// TIA Portal project "Erronka3 Igogailua" (V15.1)

(* hardware
DEVICE "S7-1200 station_1"  S7-1200 Station
   slot 0: "Rack_0"  S7-1200 Rack  Rack  V1.0
   slot 1: "PLC_1"  CPU 1214C AC/DC/Rly  6ES7 214-1BG40-0XB0  V4.2
*)

// ===== PLC "PLC_1"  CPU 1214C AC/DC/Rly =====

VAR_GLOBAL   // PLC tag table "Etapak"
   "Etapa0" AT %M16.0 : Bool;
   "Etapa1" AT %M16.1 : Bool;
   "Etapa2" AT %M16.2 : Bool;
   "Etapa3" AT %M16.3 : Bool;
   "Etapa4" AT %M16.4 : Bool;
   "Etapa5" AT %M16.5 : Bool;
   "Etapa6" AT %M16.6 : Bool;
   "Etapa3.1" AT %M17.0 : Bool;
   "Etapa10" AT %M17.1 : Bool;
   "Etapa11" AT %M17.2 : Bool;
   "Etapa12" AT %M17.3 : Bool;
   "Etapa13" AT %M17.4 : Bool;
   "Etapa14" AT %M17.5 : Bool;
   "Etapa11.1" AT %M17.6 : Bool;
   "Etapa40" AT %M17.7 : Bool;
   "Etapa41" AT %M18.0 : Bool;
   "Etapa42" AT %M18.1 : Bool;
   "Etapa43" AT %M18.2 : Bool;
   "Etapa44" AT %M18.3 : Bool;
   "Etapa50" AT %M18.4 : Bool;
   "Etapa51" AT %M18.5 : Bool;
   "Etapa52" AT %M18.6 : Bool;
   "Etapa53" AT %M18.7 : Bool;
   "Etapa54" AT %M19.0 : Bool;
   "Etapa60" AT %M19.1 : Bool;
   "Etapa61" AT %M19.2 : Bool;
END_VAR

VAR_GLOBAL   // PLC tag table "Irterak"
   "M1Subir" AT %Q0.0 : Bool;
   "M2Abrir" AT %Q0.1 : Bool;
   "M1Bajar" AT %Q0.2 : Bool;
   "M2Cerrar" AT %Q0.3 : Bool;
   "0Sube" AT %Q0.4 : Bool;
   "0Baja" AT %Q0.5 : Bool;
   "1Sube" AT %Q0.6 : Bool;
   "1Baja" AT %Q0.7 : Bool;
   "ASube" AT %Q1.0 : Bool;
   "ABaja" AT %Q1.1 : Bool;
   "M1Subir_10" AT %Q1.2 : Bool;
END_VAR

VAR_GLOBAL   // PLC tag table "Sarrerak"
   "FC0" AT %I0.0 : Bool;
   "FC1" AT %I0.1 : Bool;
   "PF0" AT %I0.2 : Bool;
   "PF1" AT %I0.3 : Bool;
   "PD1" AT %I0.4 : Bool;
   "PD0" AT %I0.5 : Bool;
   "PA" AT %I0.6 : Bool;
   "F" AT %I0.7 : Bool;
   "M" AT %I1.0 : Bool;
   "SCP" AT %I1.1 : Bool;
   "SAP" AT %I1.2 : Bool;
   "PE" AT %I1.3 : Bool;
END_VAR

// folder: System blocks/Program resources

DATA_BLOCK "Temporizador1"   // DB1
{ S7_Optimized_Access := 'TRUE' }
AUTHOR : Simatic
FAMILY : IEC
NAME : IEC_TMR
VERSION : 1.0
// stored: InstanceOfName IEC_TIMER
"IEC_TIMER"
BEGIN
END_DATA_BLOCK

// folder: (top level)

FUNCTION "Grafcet" : Void   // FC1, LAD
{ S7_Optimized_Access := 'TRUE' }
VERSION : 0.1
BEGIN

REGION Network 1: Activar etapa 1
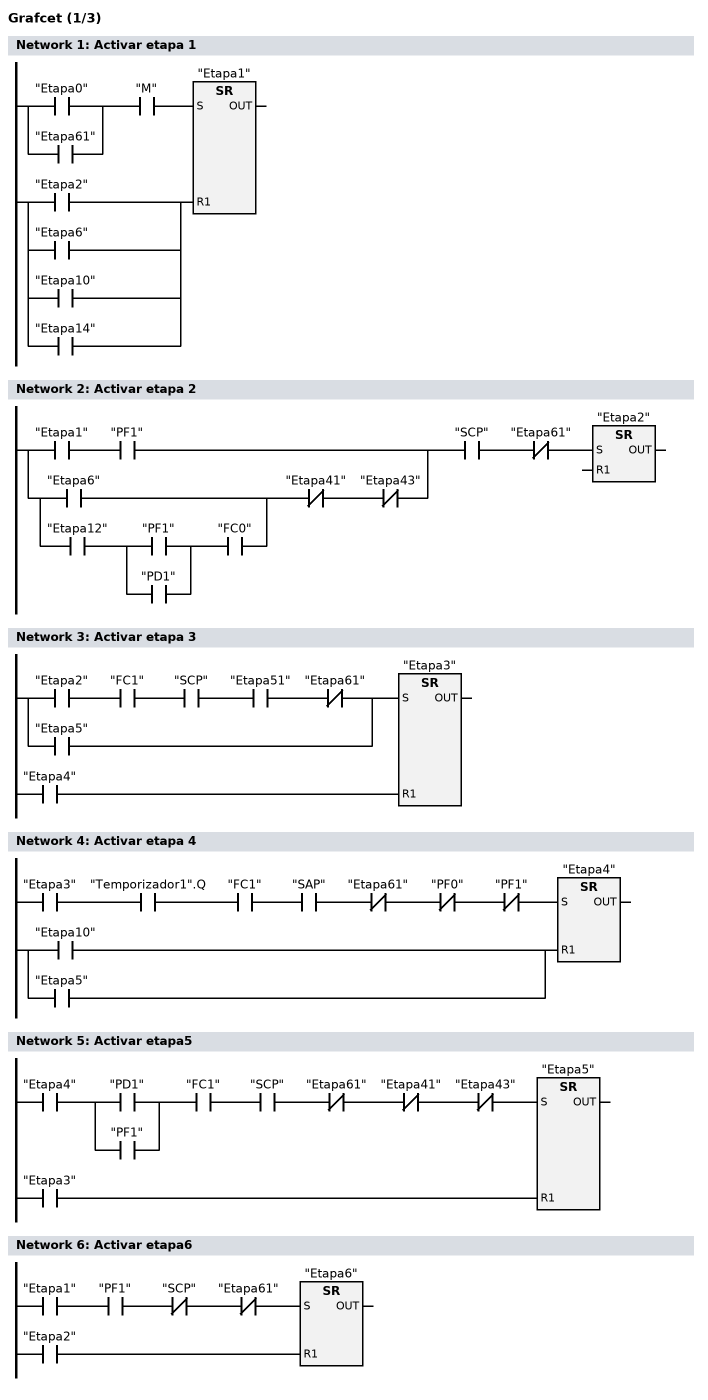
   RUNG wire#powerrail
      Contact( "Etapa0" )
      wire#w1
      Contact( "M" )
      S_SR(operand := "Etapa1", r1 := wire#w2)
   END_RUNG
   RUNG wire#powerrail
      Contact( "Etapa61" )
   END_RUNG wire#w1
   RUNG wire#powerrail
      Contact( "Etapa2" )
   END_RUNG wire#w2
   RUNG wire#powerrail
      Contact( "Etapa6" )
   END_RUNG wire#w2
   RUNG wire#powerrail
      Contact( "Etapa10" )
   END_RUNG wire#w2
   RUNG wire#powerrail
      Contact( "Etapa14" )
   END_RUNG wire#w2
   // the same network as SCL:
   IF ("Etapa0" OR "Etapa61") AND "M" THEN
       "Etapa1" := TRUE;   // SR flip-flop
   END_IF;
   IF "Etapa2" OR "Etapa6" OR "Etapa10" OR "Etapa14" THEN "Etapa1" := FALSE; END_IF;
END_REGION

REGION Network 2: Activar etapa 2
   RUNG wire#powerrail
      Contact( "Etapa1" )
      Contact( "PF1" )
      wire#w1
      Contact( "SCP" )
      I_Contact( "Etapa61" )
      S_SR(operand := "Etapa2", r1 :=)
   END_RUNG
   RUNG wire#powerrail
      Contact( "Etapa6" )
      wire#w2
      I_Contact( "Etapa41" )
      I_Contact( "Etapa43" )
   END_RUNG wire#w1
   RUNG wire#powerrail
      Contact( "Etapa12" )
      wire#w3
      Contact( "PF1" )
      wire#w4
      Contact( "FC0" )
   END_RUNG wire#w2
   RUNG wire#w3
      Contact( "PD1" )
   END_RUNG wire#w4
   // the same network as SCL:
   IF (("Etapa1" AND "PF1") OR (("Etapa6" OR ("Etapa12" AND ("PF1" OR "PD1") AND "FC0")) AND NOT "Etapa41" AND NOT "Etapa43")) AND "SCP" AND NOT "Etapa61" THEN
       "Etapa2" := TRUE;   // SR flip-flop
   END_IF;
END_REGION

REGION Network 3: Activar etapa 3
   RUNG wire#powerrail
      Contact( "Etapa2" )
      Contact( "FC1" )
      Contact( "SCP" )
      Contact( "Etapa51" )
      I_Contact( "Etapa61" )
      wire#w1
      S_SR(operand := "Etapa3", r1 := wire#w2)
   END_RUNG
   RUNG wire#powerrail
      Contact( "Etapa5" )
   END_RUNG wire#w1
   RUNG wire#powerrail
      Contact( "Etapa4" )
   END_RUNG wire#w2
   // the same network as SCL:
   IF ("Etapa2" AND "FC1" AND "SCP" AND "Etapa51" AND NOT "Etapa61") OR "Etapa5" THEN
       "Etapa3" := TRUE;   // SR flip-flop
   END_IF;
   IF "Etapa4" THEN "Etapa3" := FALSE; END_IF;
END_REGION

REGION Network 4: Activar etapa 4
   RUNG wire#powerrail
      Contact( "Etapa3" )
      Contact( "Temporizador1".Q )
      Contact( "FC1" )
      Contact( "SAP" )
      I_Contact( "Etapa61" )
      I_Contact( "PF0" )
      I_Contact( "PF1" )
      S_SR(operand := "Etapa4", r1 := wire#w1)
   END_RUNG
   RUNG wire#powerrail
      Contact( "Etapa10" )
   END_RUNG wire#w1
   RUNG wire#powerrail
      Contact( "Etapa5" )
   END_RUNG wire#w1
   // the same network as SCL:
   IF "Etapa3" AND "Temporizador1".Q AND "FC1" AND "SAP" AND NOT "Etapa61" AND NOT "PF0" AND NOT "PF1" THEN
       "Etapa4" := TRUE;   // SR flip-flop
   END_IF;
   IF "Etapa10" OR "Etapa5" THEN "Etapa4" := FALSE; END_IF;
END_REGION

REGION Network 5: Activar etapa5
   RUNG wire#powerrail
      Contact( "Etapa4" )
      wire#w1
      Contact( "PD1" )
      wire#w2
      Contact( "FC1" )
      Contact( "SCP" )
      I_Contact( "Etapa61" )
      I_Contact( "Etapa41" )
      I_Contact( "Etapa43" )
      S_SR(operand := "Etapa5", r1 := wire#w3)
   END_RUNG
   RUNG wire#w1
      Contact( "PF1" )
   END_RUNG wire#w2
   RUNG wire#powerrail
      Contact( "Etapa3" )
   END_RUNG wire#w3
   // the same network as SCL:
   IF "Etapa4" AND ("PD1" OR "PF1") AND "FC1" AND "SCP" AND NOT "Etapa61" AND NOT "Etapa41" AND NOT "Etapa43" THEN
       "Etapa5" := TRUE;   // SR flip-flop
   END_IF;
   IF "Etapa3" THEN "Etapa5" := FALSE; END_IF;
END_REGION

REGION Network 6: Activar etapa6
   RUNG wire#powerrail
      Contact( "Etapa1" )
      Contact( "PF1" )
      I_Contact( "SCP" )
      I_Contact( "Etapa61" )
      S_SR(operand := "Etapa6", r1 := wire#w1)
   END_RUNG
   RUNG wire#powerrail
      Contact( "Etapa2" )
   END_RUNG wire#w1
   // the same network as SCL:
   IF "Etapa1" AND "PF1" AND NOT "SCP" AND NOT "Etapa61" THEN
       "Etapa6" := TRUE;   // SR flip-flop
   END_IF;
   IF "Etapa2" THEN "Etapa6" := FALSE; END_IF;
END_REGION

REGION Network 7: Activar etapa3.1
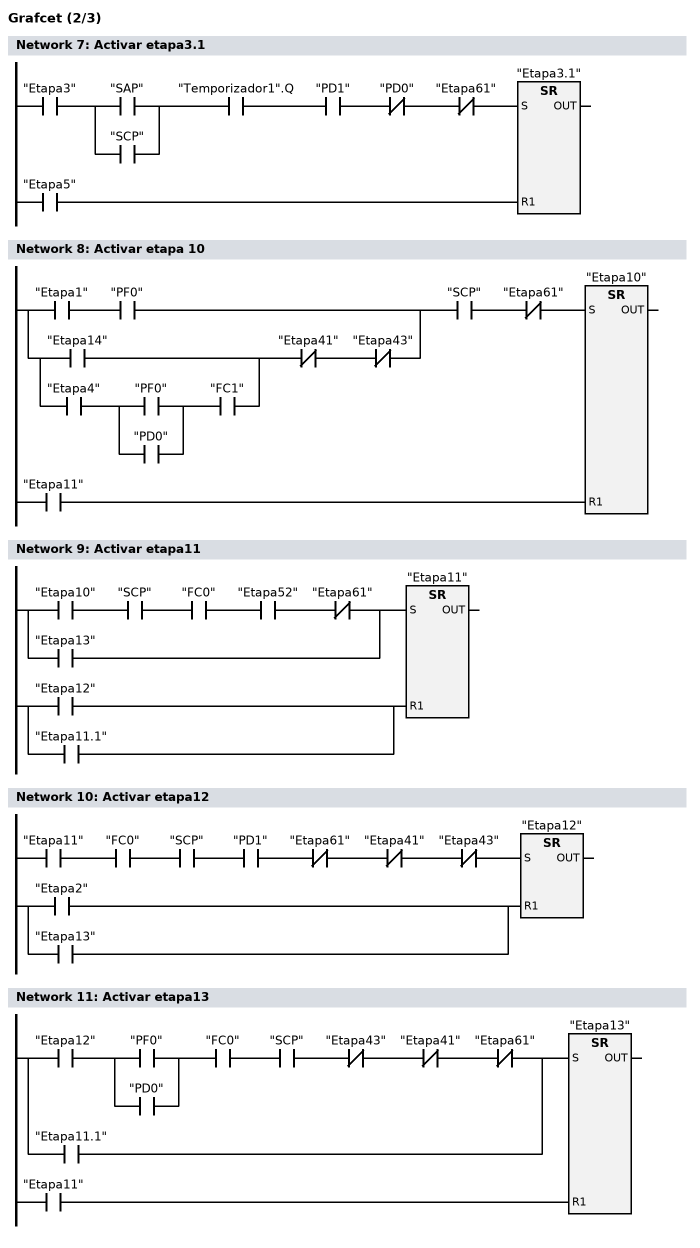
   RUNG wire#powerrail
      Contact( "Etapa3" )
      wire#w1
      Contact( "SAP" )
      wire#w2
      Contact( "Temporizador1".Q )
      Contact( "PD1" )
      I_Contact( "PD0" )
      I_Contact( "Etapa61" )
      S_SR(operand := "Etapa3.1", r1 := wire#w3)
   END_RUNG
   RUNG wire#w1
      Contact( "SCP" )
   END_RUNG wire#w2
   RUNG wire#powerrail
      Contact( "Etapa5" )
   END_RUNG wire#w3
   // the same network as SCL:
   IF "Etapa3" AND ("SAP" OR "SCP") AND "Temporizador1".Q AND "PD1" AND NOT "PD0" AND NOT "Etapa61" THEN
       "Etapa3.1" := TRUE;   // SR flip-flop
   END_IF;
   IF "Etapa5" THEN "Etapa3.1" := FALSE; END_IF;
END_REGION

REGION Network 8: Activar etapa 10
   RUNG wire#powerrail
      Contact( "Etapa1" )
      Contact( "PF0" )
      wire#w1
      Contact( "SCP" )
      I_Contact( "Etapa61" )
      S_SR(operand := "Etapa10", r1 := wire#w5)
   END_RUNG
   RUNG wire#powerrail
      Contact( "Etapa14" )
      wire#w2
      I_Contact( "Etapa41" )
      I_Contact( "Etapa43" )
   END_RUNG wire#w1
   RUNG wire#powerrail
      Contact( "Etapa4" )
      wire#w3
      Contact( "PF0" )
      wire#w4
      Contact( "FC1" )
   END_RUNG wire#w2
   RUNG wire#w3
      Contact( "PD0" )
   END_RUNG wire#w4
   RUNG wire#powerrail
      Contact( "Etapa11" )
   END_RUNG wire#w5
   // the same network as SCL:
   IF (("Etapa1" AND "PF0") OR (("Etapa14" OR ("Etapa4" AND ("PF0" OR "PD0") AND "FC1")) AND NOT "Etapa41" AND NOT "Etapa43")) AND "SCP" AND NOT "Etapa61" THEN
       "Etapa10" := TRUE;   // SR flip-flop
   END_IF;
   IF "Etapa11" THEN "Etapa10" := FALSE; END_IF;
END_REGION

REGION Network 9: Activar etapa11
   RUNG wire#powerrail
      Contact( "Etapa10" )
      Contact( "SCP" )
      Contact( "FC0" )
      Contact( "Etapa52" )
      I_Contact( "Etapa61" )
      wire#w1
      S_SR(operand := "Etapa11", r1 := wire#w2)
   END_RUNG
   RUNG wire#powerrail
      Contact( "Etapa13" )
   END_RUNG wire#w1
   RUNG wire#powerrail
      Contact( "Etapa12" )
   END_RUNG wire#w2
   RUNG wire#powerrail
      Contact( "Etapa11.1" )
   END_RUNG wire#w2
   // the same network as SCL:
   IF ("Etapa10" AND "SCP" AND "FC0" AND "Etapa52" AND NOT "Etapa61") OR "Etapa13" THEN
       "Etapa11" := TRUE;   // SR flip-flop
   END_IF;
   IF "Etapa12" OR "Etapa11.1" THEN "Etapa11" := FALSE; END_IF;
END_REGION

REGION Network 10: Activar etapa12
   RUNG wire#powerrail
      Contact( "Etapa11" )
      Contact( "FC0" )
      Contact( "SCP" )
      Contact( "PD1" )
      I_Contact( "Etapa61" )
      I_Contact( "Etapa41" )
      I_Contact( "Etapa43" )
      S_SR(operand := "Etapa12", r1 := wire#w1)
   END_RUNG
   RUNG wire#powerrail
      Contact( "Etapa2" )
   END_RUNG wire#w1
   RUNG wire#powerrail
      Contact( "Etapa13" )
   END_RUNG wire#w1
   // the same network as SCL:
   IF "Etapa11" AND "FC0" AND "SCP" AND "PD1" AND NOT "Etapa61" AND NOT "Etapa41" AND NOT "Etapa43" THEN
       "Etapa12" := TRUE;   // SR flip-flop
   END_IF;
   IF "Etapa2" OR "Etapa13" THEN "Etapa12" := FALSE; END_IF;
END_REGION

REGION Network 11: Activar etapa13
   RUNG wire#powerrail
      Contact( "Etapa12" )
      wire#w1
      Contact( "PF0" )
      wire#w2
      Contact( "FC0" )
      Contact( "SCP" )
      I_Contact( "Etapa43" )
      I_Contact( "Etapa41" )
      I_Contact( "Etapa61" )
      wire#w3
      S_SR(operand := "Etapa13", r1 := wire#w4)
   END_RUNG
   RUNG wire#w1
      Contact( "PD0" )
   END_RUNG wire#w2
   RUNG wire#powerrail
      Contact( "Etapa11.1" )
   END_RUNG wire#w3
   RUNG wire#powerrail
      Contact( "Etapa11" )
   END_RUNG wire#w4
   // the same network as SCL:
   IF ("Etapa12" AND ("PF0" OR "PD0") AND "FC0" AND "SCP" AND NOT "Etapa43" AND NOT "Etapa41" AND NOT "Etapa61") OR "Etapa11.1" THEN
       "Etapa13" := TRUE;   // SR flip-flop
   END_IF;
   IF "Etapa11" THEN "Etapa13" := FALSE; END_IF;
END_REGION

REGION Network 12: Activar etapa11.1
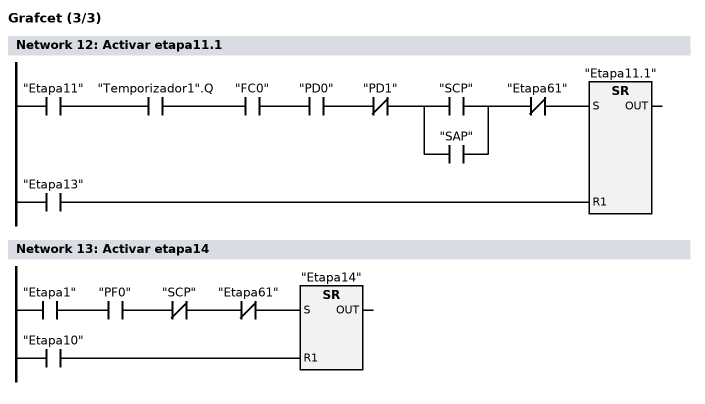
   RUNG wire#powerrail
      Contact( "Etapa11" )
      Contact( "Temporizador1".Q )
      Contact( "FC0" )
      Contact( "PD0" )
      I_Contact( "PD1" )
      wire#w1
      Contact( "SCP" )
      wire#w2
      I_Contact( "Etapa61" )
      S_SR(operand := "Etapa11.1", r1 := wire#w3)
   END_RUNG
   RUNG wire#w1
      Contact( "SAP" )
   END_RUNG wire#w2
   RUNG wire#powerrail
      Contact( "Etapa13" )
   END_RUNG wire#w3
   // the same network as SCL:
   IF "Etapa11" AND "Temporizador1".Q AND "FC0" AND "PD0" AND NOT "PD1" AND ("SCP" OR "SAP") AND NOT "Etapa61" THEN
       "Etapa11.1" := TRUE;   // SR flip-flop
   END_IF;
   IF "Etapa13" THEN "Etapa11.1" := FALSE; END_IF;
END_REGION

REGION Network 13: Activar etapa14
   RUNG wire#powerrail
      Contact( "Etapa1" )
      Contact( "PF0" )
      I_Contact( "SCP" )
      I_Contact( "Etapa61" )
      S_SR(operand := "Etapa14", r1 := wire#w1)
   END_RUNG
   RUNG wire#powerrail
      Contact( "Etapa10" )
   END_RUNG wire#w1
   // the same network as SCL:
   IF "Etapa1" AND "PF0" AND NOT "SCP" AND NOT "Etapa61" THEN
       "Etapa14" := TRUE;   // SR flip-flop
   END_IF;
   IF "Etapa10" THEN "Etapa14" := FALSE; END_IF;
END_REGION
END_FUNCTION

FUNCTION "Subrutina 40" : Void   // FC2, LAD
{ S7_Optimized_Access := 'TRUE' }
VERSION : 0.1
BEGIN

REGION Network 1: Subrutina 40
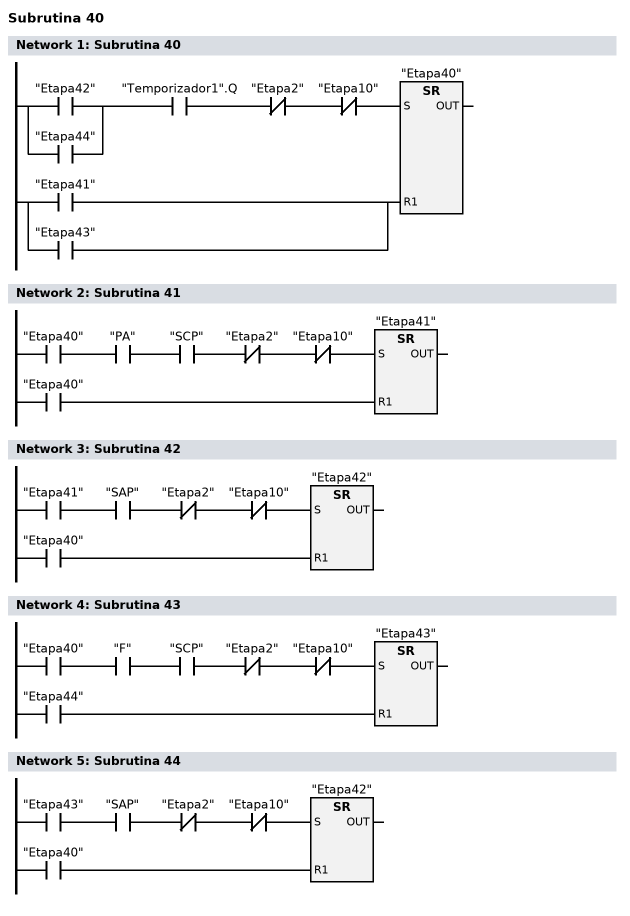
   RUNG wire#powerrail
      Contact( "Etapa42" )
      wire#w1
      Contact( "Temporizador1".Q )
      I_Contact( "Etapa2" )
      I_Contact( "Etapa10" )
      S_SR(operand := "Etapa40", r1 := wire#w2)
   END_RUNG
   RUNG wire#powerrail
      Contact( "Etapa44" )
   END_RUNG wire#w1
   RUNG wire#powerrail
      Contact( "Etapa41" )
   END_RUNG wire#w2
   RUNG wire#powerrail
      Contact( "Etapa43" )
   END_RUNG wire#w2
   // the same network as SCL:
   IF ("Etapa42" OR "Etapa44") AND "Temporizador1".Q AND NOT "Etapa2" AND NOT "Etapa10" THEN
       "Etapa40" := TRUE;   // SR flip-flop
   END_IF;
   IF "Etapa41" OR "Etapa43" THEN "Etapa40" := FALSE; END_IF;
END_REGION

REGION Network 2: Subrutina 41
   RUNG wire#powerrail
      Contact( "Etapa40" )
      Contact( "PA" )
      Contact( "SCP" )
      I_Contact( "Etapa2" )
      I_Contact( "Etapa10" )
      S_SR(operand := "Etapa41", r1 := wire#w1)
   END_RUNG
   RUNG wire#powerrail
      Contact( "Etapa40" )
   END_RUNG wire#w1
   // the same network as SCL:
   IF "Etapa40" AND "PA" AND "SCP" AND NOT "Etapa2" AND NOT "Etapa10" THEN
       "Etapa41" := TRUE;   // SR flip-flop
   END_IF;
   IF "Etapa40" THEN "Etapa41" := FALSE; END_IF;
END_REGION

REGION Network 3: Subrutina 42
   RUNG wire#powerrail
      Contact( "Etapa41" )
      Contact( "SAP" )
      I_Contact( "Etapa2" )
      I_Contact( "Etapa10" )
      S_SR(operand := "Etapa42", r1 := wire#w1)
   END_RUNG
   RUNG wire#powerrail
      Contact( "Etapa40" )
   END_RUNG wire#w1
   // the same network as SCL:
   IF "Etapa41" AND "SAP" AND NOT "Etapa2" AND NOT "Etapa10" THEN
       "Etapa42" := TRUE;   // SR flip-flop
   END_IF;
   IF "Etapa40" THEN "Etapa42" := FALSE; END_IF;
END_REGION

REGION Network 4: Subrutina 43
   RUNG wire#powerrail
      Contact( "Etapa40" )
      Contact( "F" )
      Contact( "SCP" )
      I_Contact( "Etapa2" )
      I_Contact( "Etapa10" )
      S_SR(operand := "Etapa43", r1 := wire#w1)
   END_RUNG
   RUNG wire#powerrail
      Contact( "Etapa44" )
   END_RUNG wire#w1
   // the same network as SCL:
   IF "Etapa40" AND "F" AND "SCP" AND NOT "Etapa2" AND NOT "Etapa10" THEN
       "Etapa43" := TRUE;   // SR flip-flop
   END_IF;
   IF "Etapa44" THEN "Etapa43" := FALSE; END_IF;
END_REGION

REGION Network 5: Subrutina 44
   RUNG wire#powerrail
      Contact( "Etapa43" )
      Contact( "SAP" )
      I_Contact( "Etapa2" )
      I_Contact( "Etapa10" )
      S_SR(operand := "Etapa42", r1 := wire#w1)
   END_RUNG
   RUNG wire#powerrail
      Contact( "Etapa40" )
   END_RUNG wire#w1
   // the same network as SCL:
   IF "Etapa43" AND "SAP" AND NOT "Etapa2" AND NOT "Etapa10" THEN
       "Etapa42" := TRUE;   // SR flip-flop
   END_IF;
   IF "Etapa40" THEN "Etapa42" := FALSE; END_IF;
END_REGION
END_FUNCTION

FUNCTION "Grafcet Irterak" : Void   // FC3, LAD
{ S7_Optimized_Access := 'TRUE' }
VERSION : 0.1
BEGIN

REGION Network 1: Etapa1
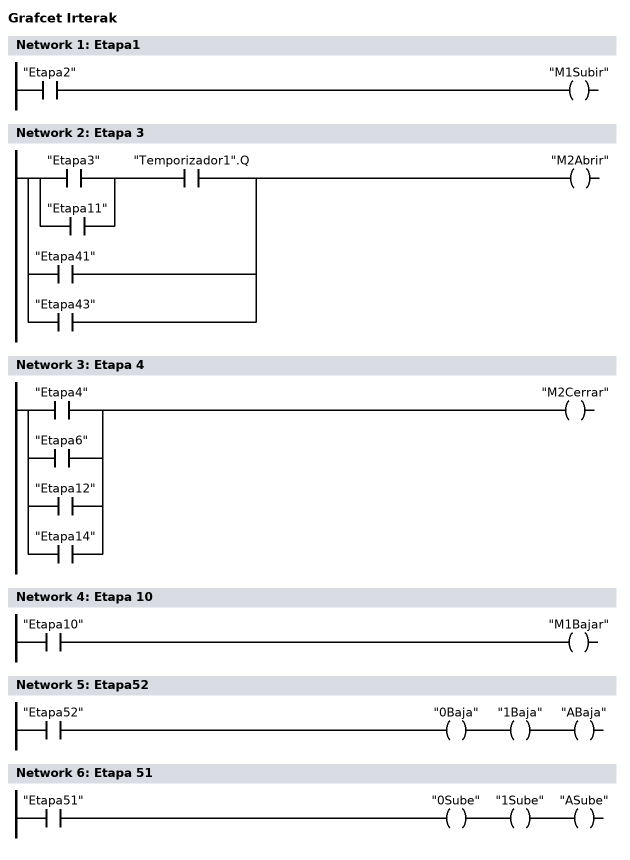
   RUNG wire#powerrail
      Contact( "Etapa2" )
      Coil( "M1Subir" )
   END_RUNG
   // the same network as SCL:
   "M1Subir" := "Etapa2";
END_REGION

REGION Network 2: Etapa 3
   RUNG wire#powerrail
      Contact( "Etapa3" )
      wire#w1
      Contact( "Temporizador1".Q )
      wire#w2
      Coil( "M2Abrir" )
   END_RUNG
   RUNG wire#powerrail
      Contact( "Etapa11" )
   END_RUNG wire#w1
   RUNG wire#powerrail
      Contact( "Etapa41" )
   END_RUNG wire#w2
   RUNG wire#powerrail
      Contact( "Etapa43" )
   END_RUNG wire#w2
   // the same network as SCL:
   "M2Abrir" := (("Etapa3" OR "Etapa11") AND "Temporizador1".Q) OR "Etapa41" OR "Etapa43";
END_REGION

REGION Network 3: Etapa 4
   RUNG wire#powerrail
      Contact( "Etapa4" )
      wire#w1
      Coil( "M2Cerrar" )
   END_RUNG
   RUNG wire#powerrail
      Contact( "Etapa6" )
   END_RUNG wire#w1
   RUNG wire#powerrail
      Contact( "Etapa12" )
   END_RUNG wire#w1
   RUNG wire#powerrail
      Contact( "Etapa14" )
   END_RUNG wire#w1
   // the same network as SCL:
   "M2Cerrar" := "Etapa4" OR "Etapa6" OR "Etapa12" OR "Etapa14";
END_REGION

REGION Network 4: Etapa 10
   RUNG wire#powerrail
      Contact( "Etapa10" )
      Coil( "M1Bajar" )
   END_RUNG
   // the same network as SCL:
   "M1Bajar" := "Etapa10";
END_REGION

REGION Network 5: Etapa52
   RUNG wire#powerrail
      Contact( "Etapa52" )
      Coil( "0Baja" )
      Coil( "1Baja" )
      Coil( "ABaja" )
   END_RUNG
   // the same network as SCL:
   "0Baja" := "Etapa52";
   "1Baja" := "Etapa52";
   "ABaja" := "Etapa52";
END_REGION

REGION Network 6: Etapa 51
   RUNG wire#powerrail
      Contact( "Etapa51" )
      Coil( "0Sube" )
      Coil( "1Sube" )
      Coil( "ASube" )
   END_RUNG
   // the same network as SCL:
   "0Sube" := "Etapa51";
   "1Sube" := "Etapa51";
   "ASube" := "Etapa51";
END_REGION
END_FUNCTION

FUNCTION "Subrutina 50" : Void   // FC4, LAD
{ S7_Optimized_Access := 'TRUE' }
VERSION : 0.1
BEGIN

REGION Network 1: Subrutina 50
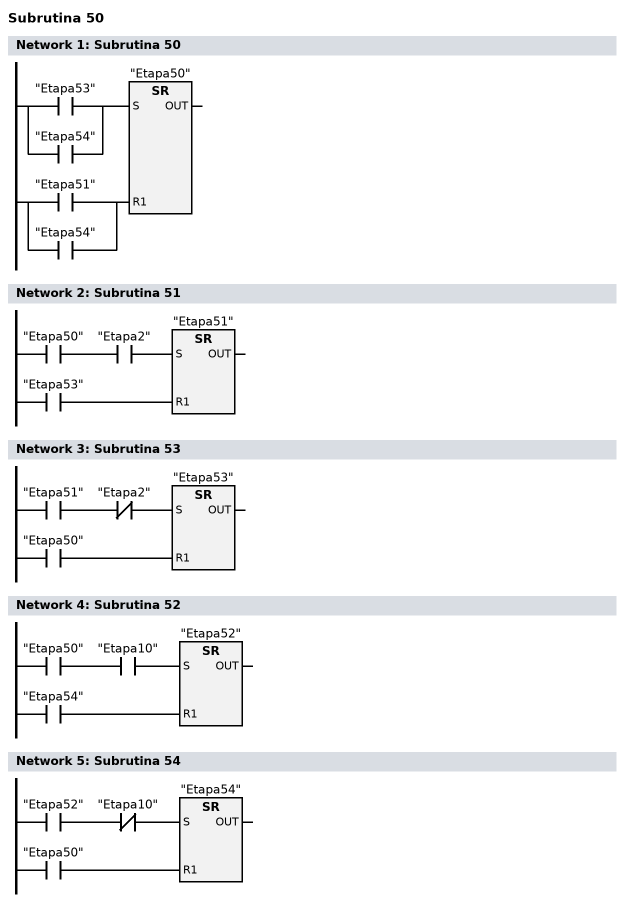
   RUNG wire#powerrail
      Contact( "Etapa53" )
      wire#w1
      S_SR(operand := "Etapa50", r1 := wire#w2)
   END_RUNG
   RUNG wire#powerrail
      Contact( "Etapa54" )
   END_RUNG wire#w1
   RUNG wire#powerrail
      Contact( "Etapa51" )
   END_RUNG wire#w2
   RUNG wire#powerrail
      Contact( "Etapa54" )
   END_RUNG wire#w2
   // the same network as SCL:
   IF "Etapa53" OR "Etapa54" THEN
       "Etapa50" := TRUE;   // SR flip-flop
   END_IF;
   IF "Etapa51" OR "Etapa54" THEN "Etapa50" := FALSE; END_IF;
END_REGION

REGION Network 2: Subrutina 51
   RUNG wire#powerrail
      Contact( "Etapa50" )
      Contact( "Etapa2" )
      S_SR(operand := "Etapa51", r1 := wire#w1)
   END_RUNG
   RUNG wire#powerrail
      Contact( "Etapa53" )
   END_RUNG wire#w1
   // the same network as SCL:
   IF "Etapa50" AND "Etapa2" THEN
       "Etapa51" := TRUE;   // SR flip-flop
   END_IF;
   IF "Etapa53" THEN "Etapa51" := FALSE; END_IF;
END_REGION

REGION Network 3: Subrutina 53
   RUNG wire#powerrail
      Contact( "Etapa51" )
      I_Contact( "Etapa2" )
      S_SR(operand := "Etapa53", r1 := wire#w1)
   END_RUNG
   RUNG wire#powerrail
      Contact( "Etapa50" )
   END_RUNG wire#w1
   // the same network as SCL:
   IF "Etapa51" AND NOT "Etapa2" THEN
       "Etapa53" := TRUE;   // SR flip-flop
   END_IF;
   IF "Etapa50" THEN "Etapa53" := FALSE; END_IF;
END_REGION

REGION Network 4: Subrutina 52
   RUNG wire#powerrail
      Contact( "Etapa50" )
      Contact( "Etapa10" )
      S_SR(operand := "Etapa52", r1 := wire#w1)
   END_RUNG
   RUNG wire#powerrail
      Contact( "Etapa54" )
   END_RUNG wire#w1
   // the same network as SCL:
   IF "Etapa50" AND "Etapa10" THEN
       "Etapa52" := TRUE;   // SR flip-flop
   END_IF;
   IF "Etapa54" THEN "Etapa52" := FALSE; END_IF;
END_REGION

REGION Network 5: Subrutina 54
   RUNG wire#powerrail
      Contact( "Etapa52" )
      I_Contact( "Etapa10" )
      S_SR(operand := "Etapa54", r1 := wire#w1)
   END_RUNG
   RUNG wire#powerrail
      Contact( "Etapa50" )
   END_RUNG wire#w1
   // the same network as SCL:
   IF "Etapa52" AND NOT "Etapa10" THEN
       "Etapa54" := TRUE;   // SR flip-flop
   END_IF;
   IF "Etapa50" THEN "Etapa54" := FALSE; END_IF;
END_REGION
END_FUNCTION

FUNCTION "Subrutina 60" : Void   // FC5, LAD
{ S7_Optimized_Access := 'TRUE' }
VERSION : 0.1
BEGIN

REGION Network 1: Subrutina61
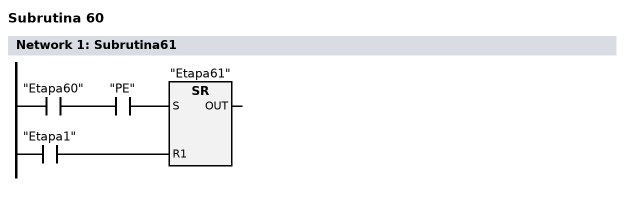
   RUNG wire#powerrail
      Contact( "Etapa60" )
      Contact( "PE" )
      S_SR(operand := "Etapa61", r1 := wire#w1)
   END_RUNG
   RUNG wire#powerrail
      Contact( "Etapa1" )
   END_RUNG wire#w1
   // the same network as SCL:
   IF "Etapa60" AND "PE" THEN
       "Etapa61" := TRUE;   // SR flip-flop
   END_IF;
   IF "Etapa1" THEN "Etapa61" := FALSE; END_IF;
END_REGION
END_FUNCTION

FUNCTION "Temporizador" : Void   // FC6, LAD
{ S7_Optimized_Access := 'TRUE' }
VERSION : 0.1
BEGIN

REGION Network 1: Hau da temporizadorea
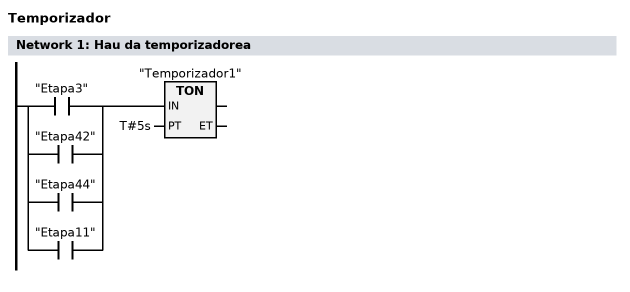
   "Temporizador1".TON(IN := "Etapa3" OR "Etapa42" OR "Etapa44" OR "Etapa11", PT := T#5s);
END_REGION
END_FUNCTION

ORGANIZATION_BLOCK "Main"   // OB1, LAD, ProgramCycle
TITLE = "Main Program Sweep (Cycle)"
{ S7_Optimized_Access := 'TRUE' }
VERSION : 0.1
   VAR_INPUT
      Initial_Call : Bool;   // Initial call of this OB
      Remanence : Bool;   // =True, if remanent data are available
   END_VAR
BEGIN

REGION Network 1: Grafcet
   // Llamamos a la funcion grafcet la cual esta separada del main y contiene todos los segmentos para declarar las etapas
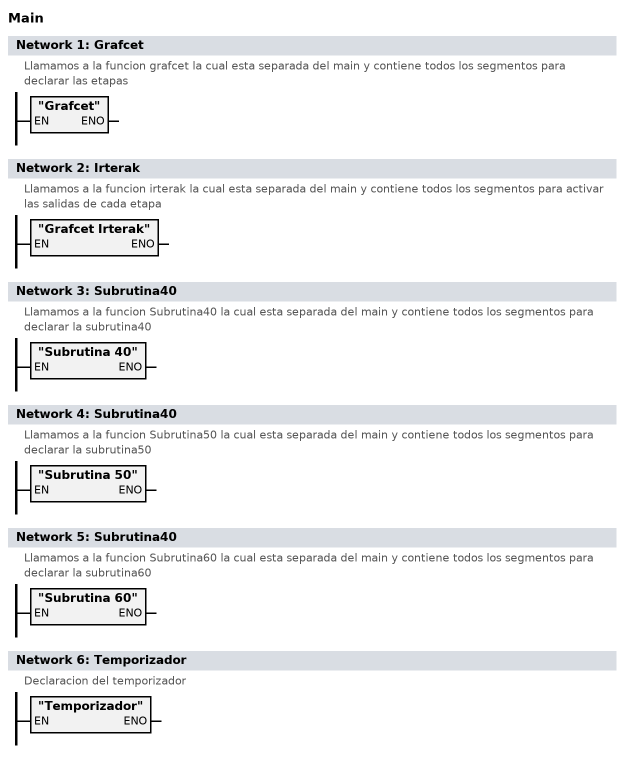
   RUNG wire#powerrail
      "Grafcet"()
   END_RUNG
   // the same network as SCL:
   "Grafcet"();
END_REGION

REGION Network 2: Irterak
   // Llamamos a la funcion irterak la cual esta separada del main y contiene todos los segmentos para activar las salidas de cada etapa
   RUNG wire#powerrail
      "Grafcet Irterak"()
   END_RUNG
   // the same network as SCL:
   "Grafcet Irterak"();
END_REGION

REGION Network 3: Subrutina40
   // Llamamos a la funcion Subrutina40 la cual esta separada del main y contiene todos los segmentos para declarar la subrutina40
   RUNG wire#powerrail
      "Subrutina 40"()
   END_RUNG
   // the same network as SCL:
   "Subrutina 40"();
END_REGION

REGION Network 4: Subrutina40
   // Llamamos a la funcion Subrutina50 la cual esta separada del main y contiene todos los segmentos para declarar la subrutina50
   RUNG wire#powerrail
      "Subrutina 50"()
   END_RUNG
   // the same network as SCL:
   "Subrutina 50"();
END_REGION

REGION Network 5: Subrutina40
   // Llamamos a la funcion Subrutina60 la cual esta separada del main y contiene todos los segmentos para declarar la subrutina60
   RUNG wire#powerrail
      "Subrutina 60"()
   END_RUNG
   // the same network as SCL:
   "Subrutina 60"();
END_REGION

REGION Network 6: Temporizador
   // Declaracion del temporizador
   RUNG wire#powerrail
      "Temporizador"()
   END_RUNG
   // the same network as SCL:
   "Temporizador"();
END_REGION
END_ORGANIZATION_BLOCK

ORGANIZATION_BLOCK "Startup"   // OB100, LAD, Startup
TITLE = "Complete Restart"
{ S7_Optimized_Access := 'TRUE' }
VERSION : 0.1
   VAR_INPUT
      LostRetentive : Bool;   // True if retentive data are lost
      LostRTC : Bool;   // True if date and time are lost
   END_VAR
BEGIN

REGION Network 1
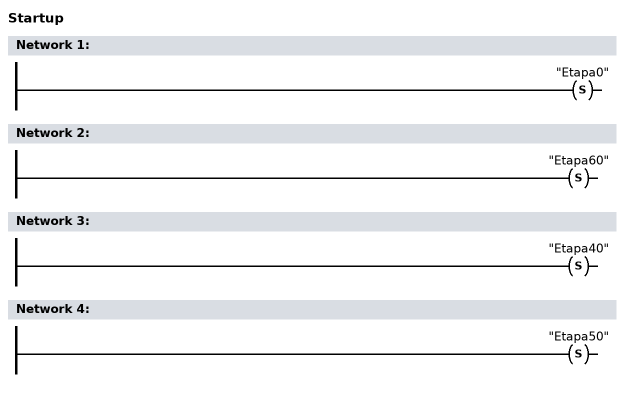
   RUNG wire#powerrail
      S_Coil( "Etapa0" )
   END_RUNG
   // the same network as SCL:
   "Etapa0" := TRUE;
END_REGION

REGION Network 2
   RUNG wire#powerrail
      S_Coil( "Etapa60" )
   END_RUNG
   // the same network as SCL:
   "Etapa60" := TRUE;
END_REGION

REGION Network 3
   RUNG wire#powerrail
      S_Coil( "Etapa40" )
   END_RUNG
   // the same network as SCL:
   "Etapa40" := TRUE;
END_REGION

REGION Network 4
   RUNG wire#powerrail
      S_Coil( "Etapa50" )
   END_RUNG
   // the same network as SCL:
   "Etapa50" := TRUE;
END_REGION
END_ORGANIZATION_BLOCK